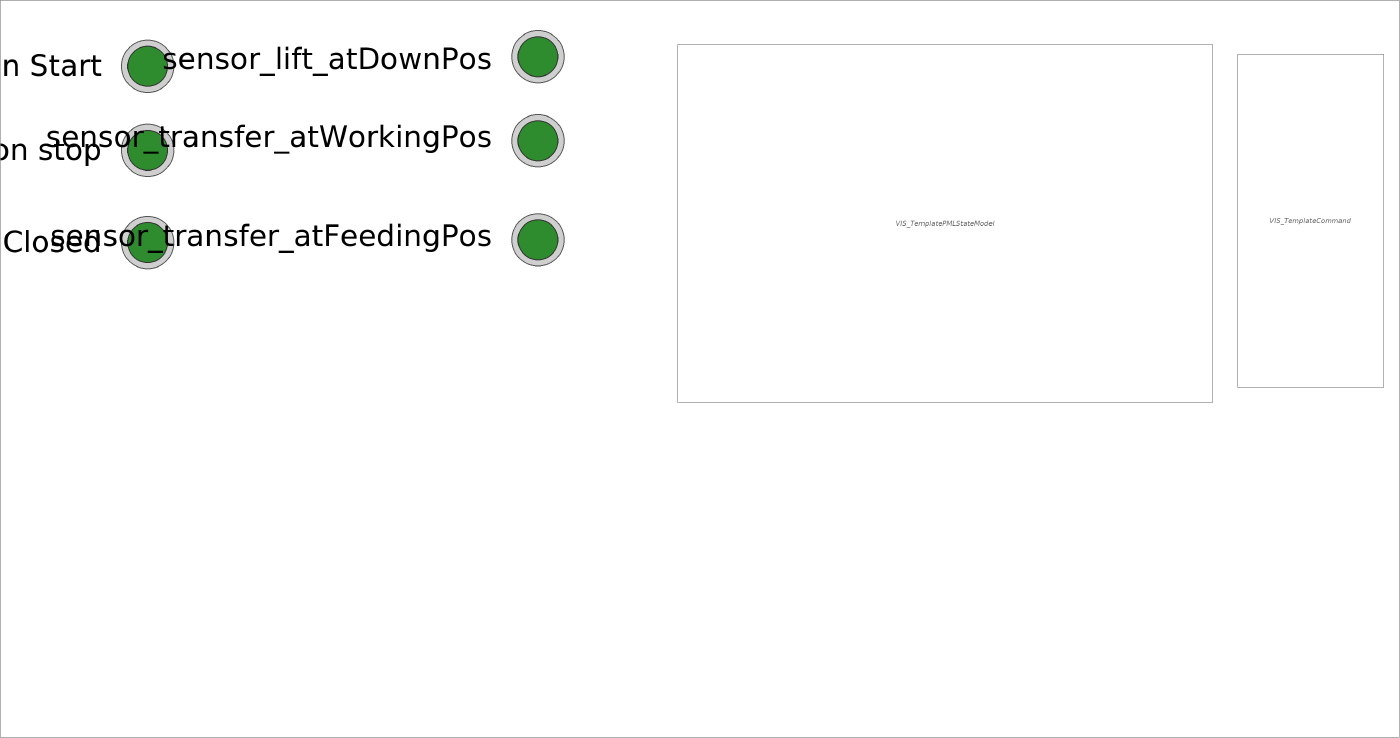
VISUALIZATION v_io_autoStore  // 2048x1080
VAR_IN_OUT
	autoStore	: FB_autoStore;
END_VAR
    Lamp1 (171,52 90x90), variable: autoStore.button_start, style: Lamp-Lamp1-Green
    Label (32,51 120x90), "Btton Start"
    Lamp1 (171,175 90x90), variable: autoStore.button_stop, style: Lamp-Lamp1-Green
    Label (32,174 120x90), "Button stop"
    Lamp1 (171,310 90x90), variable: autoStore.door_closed, style: Lamp-Lamp1-Green
    Label (32,309 120x90), "Door Closed"
    Lamp1 (742,38 90x90), variable: autoStore.sensor_lift_atDownPos, style: Lamp-Lamp1-Green
    Label (409,52 314x68), "sensor_lift_atDownPos"
    Lamp1 (742,161 90x90), variable: autoStore.sensor_transfer_atWorkingPos, style: Lamp-Lamp1-Green
    Label (339,170 384x60), "sensor_transfer_atWorkingPos"
    Lamp1 (742,306 90x90), variable: autoStore.sensor_transfer_atFeedingPos, style: Lamp-Lamp1-Green
    Label (339,315 384x60), "sensor_transfer_atFeedingPos"
    Frame (991,65 783x524)
        shows VIS_TemplatePMLStateModel(ePMLUnitMode := MAIN.fbVisu.eModeVisu, ePMLState := GVL.fb_autoStore1.eState, eStateCommand := MAIN.fbVisu.eUnitCommand)
        shows VIS_TemplatePMLStateModel()
    Frame (1810,79 214x488)
        shows VIS_TemplateCommand(eModeCommand := GVL.PackTags.Command.UnitMode, eStateCommand := GVL.PackTags1.Command.CntrlCmd, eModeStatus := GVL.PackTags.Status.UnitModeCurrent, eStateStatus := GVL.PackTags1.Status.StateCurrent, bModeChangeReq := GVL.PackTags.Command.UnitModeChangeRequest)
END_VISUALIZATION

(* stored: Version 1.1.0.1, ProductVersion 3.1.4024.12
   Visu v_io_autoStore: Id {57a8189b-b2ce-4e1d-acdd-e044e6ea38a1} *)
